// TwinCAT 3 PLC project Mbc_Tc3_Pcs
// Title: MBC TC3 PCS Library
// Company: mbc engineering GmbH
// Author: mbc engineering GmbH
// ProjectVersion: 1.2.1.1
// Description: Copyright mbc engineering GmbH Licensed under the Apache License, Version 2.0 (the "License"); you may not use this file except in compliance with the License. You may obtain a copy of the License at http://www.apache.org/licenses/LICENSE-2.0 Unless required by applicable law or agreed to in writing, software distributed under the License is distributed on an "AS IS" BASIS, WITHOUT WARRANTIES OR CONDITIONS OF ANY KIND, either express or implied. See the License for the specific language governing permissions and limitations under the License.
// ProgramVersion: 3.1.4022.2
// project tree:
//   Command/ CommandBase.TcPOU, E_CommandResultCode.TcDUT, ICommand.TcIO, ST_CommandBaseHandshake.TcDUT
//   Version/ Global_Version.TcGVL

// ---- Command/E_CommandResultCode.TcDUT
(*---------------------------------------------------------------------------
 Copyright (c) 2018 BY mbc engineering GmbH, CH-6015 Luzern
 Licensed under the Apache License, Version 2.0
-----------------------------------------------------------------------------*)
// Default Result Code of the Command
{attribute 'qualified_only'}
TYPE E_CommandResultCode :
(
	Init 			:= 0,
	Running 		:= 1,
	Done 			:= 2,
	Cancelled 		:= 3,
	StartCustom 	:= 100
) UINT;
END_TYPE

// ---- Command/ST_CommandBaseHandshake.TcDUT
(*---------------------------------------------------------------------------
 Copyright (c) 2018 BY mbc engineering GmbH, CH-6015 Luzern
 Licensed under the Apache License, Version 2.0
-----------------------------------------------------------------------------*)
// Strukture for communication with PCS in the ``CommandBase`` class
TYPE ST_CommandBaseHandshake :
STRUCT
	bExecute		: BOOL;			// Will be set to true from the PCS to start the command. When the operation is finished, the PLC will it set to false. On a long running Task, the PCS can reset to false for Abort the operation. 
	bBusy			: BOOL;			// Is True when the command is executing.
	bEnabled		: BOOL := TRUE;	// Enables a command. Only PLC writes this flag. PCS only reads this flag. 
	nResultCode		: UINT;			// Shows the operation result code of the commando state. Default Values see 'CommandResultCode' Enum Type. It is possible to set other codes!
	nProgress		: BYTE;			// Shows the optional calculated progress. The value is depend on the command implementation. (default can be 0..100%). Only necessary on long running operations.
	nSubTask		: UINT;			// Shows the optional state of long running Command Execution. It is possible to set it on own need.
END_STRUCT
END_TYPE

// ---- Version/Global_Version.TcGVL
{attribute 'TcGenerated'}
{attribute 'no-analysis'}
{attribute 'linkalways'}
// This function has been automatically generated from the project information.
VAR_GLOBAL CONSTANT
	{attribute 'const_non_replaced'}
	stLibVersion_MBC_TC3_PCS_Library : ST_LibVersion := (iMajor := 1, iMinor := 2, iBuild := 1, iRevision := 1, nFlags := 0, sVersion := '1.2.1.1');
END_VAR

// ---- Command/ICommand.TcIO
(*---------------------------------------------------------------------------
 Copyright (c) 2018 BY mbc engineering GmbH, CH-6015 Luzern
 Licensed under the Apache License, Version 2.0
-----------------------------------------------------------------------------*)
// Command interface
INTERFACE ICommand

// The method is called in each cycle to execute the funktional part and the states of the command implementation.
METHOD Call
END_METHOD

END_INTERFACE

// ---- Command/CommandBase.TcPOU
(*---------------------------------------------------------------------------
 Copyright (c) 2018 BY mbc engineering GmbH, CH-6015 Luzern
 Licensed under the Apache License, Version 2.0
-----------------------------------------------------------------------------*)
// Basic implementation of a default command class for PCS interagtion with internal structure of ``ST_CommandBaseHandshake``.
// Aditional IN and OUT parameters should be declared in the derived implementation.
FUNCTION_BLOCK PUBLIC CommandBase IMPLEMENTS ICommand
VAR_IN_OUT
	(* Use Class Properties for IN_OUT Parameters!!! *)
END_VAR
VAR
	stHandshake		: ST_CommandBaseHandshake;		// Internal variable strukture for communication with PCS.
END_VAR

// OO-Class 
Call();

// Can be used to calculate the ``stHandshake.nProgress`` and ``stHandshake.nSubTask``
METHOD PROTECTED CalculateProgress
IF stHandshake.nResultCode = E_CommandResultCode.Done THEN
	stHandshake.nProgress := 100;
END_IF
END_METHOD

// The method is called in each cycle to execute the funktional part and the states of the command implementation.
METHOD Public Call
VAR
	bInit		: BOOL;
	HEN: INT;
END_VAR
// Starting Case
stHandshake.bBusy S= bInit := (stHandshake.bExecute AND NOT stHandshake.bBusy AND stHandshake.bEnabled);
IF bInit THEN
	stHandshake.nResultCode := E_CommandResultCode.Init;
	Init();
END_IF

// Cancel by User Transition
IF (NOT stHandshake.bExecute AND stHandshake.bBusy)THEN
	Finish(E_CommandResultCode.Cancelled);	
END_IF

// Cancel State
IF (stHandshake.nResultCode = E_CommandResultCode.Cancelled)THEN
	Cancelled();
END_IF

// Running State
IF stHandshake.bExecute AND stHandshake.bBusy THEN
	
	IF Task() THEN
		// Done Transition
		Finish(E_CommandResultCode.Done);
	END_IF
END_IF

// Done State
IF (stHandshake.nResultCode = E_CommandResultCode.Done) THEN
	Done();
END_IF

CalculateProgress();
END_METHOD

// Will be called at the Cancel state when the execution is finished with the result code ``Cancelled`` or ``stHandshake.bExecute`` changes to ``false`` while ``stHandshake.bBusy`` is ```true``
METHOD PROTECTED Cancelled
;
END_METHOD

// Will be called when ``Running`` state is done and the actual state is ``Done``.
METHOD PROTECTED Done
VAR_INPUT
END_VAR
;
END_METHOD

// Can be use to finish the ``Task`` Execution with a ``nResultCode``. By using the ``Finish(E_CommandResultCode.Cancelled)`` or ``Finish(E_CommandResultCode.Done)`` calls, to the coresponding states methods ``Done`` and ``Cancelled`` will be called.  
METHOD PROTECTED Finish
VAR_INPUT
	nResultCode		: UINT;
END_VAR
stHandshake.bBusy := stHandshake.bExecute := FALSE;
stHandshake.nResultCode := nResultCode;
END_METHOD

// Will be called when ``stHandshake.bExecute`` changes to ``true`` one cycle and in the same cycle.
METHOD PROTECTED Init
VAR_INPUT
END_VAR
stHandshake.nResultCode := E_CommandResultCode.Running;
stHandshake.nProgress := 0;
stHandshake.nSubTask := 0;
END_METHOD

// Set the Progress from everywhere in the application (Regular from CalculateProgress Method)
PROPERTY PROTECTED Progress : BYTE
GET
Progress := stHandshake.nProgress;
END_GET
SET
stHandshake.nProgress := Progress;
END_SET
END_PROPERTY

// Set the SubTask Information from everywhere in the application (Regular from CalculateProgress Method)
PROPERTY PROTECTED SubTask : UINT
GET
SubTask := stHandshake.nSubTask;
END_GET
SET
stHandshake.nSubTask := SubTask;
END_SET
END_PROPERTY

// Execute the funktional part of the command implementation. Will also be executed in the same cycle ``stHandshake.bExecute`` changes to ``true`` after the ``Init`` Method
METHOD PROTECTED Task : BOOL
// Task complete if return true
Task := TRUE;
END_METHOD

END_FUNCTION_BLOCK
